FUNCTION F_DeliverType : string
VAR_INPUT
	iSample : I_Name;
END_VAR

F_DeliverType := iSample.GetType();

END_FUNCTION

(* stored: Version 1.1.0.1, ProductVersion 3.1.4024.12
   POU F_DeliverType: Id {333942c0-18d7-42a9-869b-1f478500edd9}, SpecialFunc None *)
